FUNCTION TryConvert_DWORD_TO_DWORD : BOOL
VAR_INPUT
	in : DWORD;
	out : REFERENCE TO DWORD;
END_VAR

out := in;
TryConvert_DWORD_TO_DWORD := TRUE;

END_FUNCTION

(* stored: Version 1.1.0.1, ProductVersion 3.1.4024.12
   POU TryConvert_DWORD_TO_DWORD: Id {30e05fad-2ac8-480f-a6b0-a13c8beda329}, SpecialFunc None *)
